SUBAPPLICATION mapping_AuxFunction2_IE (* Mapping for all AuxFunction2 *)
  (* Standard: 61499-2 *)
  (* Version 1.0, 2023-01-29, Franz *)
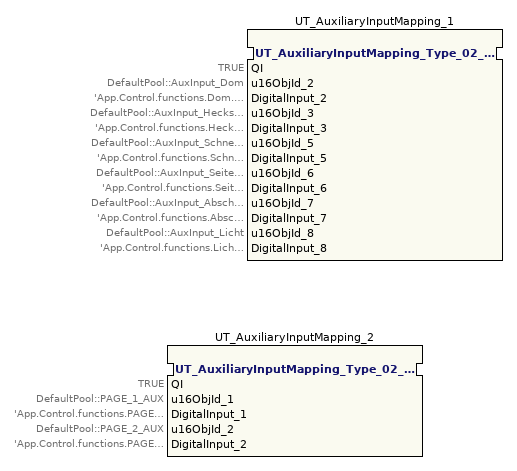
  FBS
    UT_AuxiliaryInputMapping_1 : UT_AuxiliaryInputMapping_Type_02_Bool_NonLatched_UP(QI := TRUE, u16ObjId_2 := DefaultPool::AuxInput_Dom, DigitalInput_2 := 'App.Control.functions.Dom.AuxInput', u16ObjId_3 := DefaultPool::AuxInput_Heckschieber, DigitalInput_3 := 'App.Control.functions.Heckschieber.AuxInput', u16ObjId_5 := DefaultPool::AuxInput_Schneidwerk, DigitalInput_5 := 'App.Control.functions.Schneidwerk.AuxInput', u16ObjId_6 := DefaultPool::AuxInput_Seitenschieber, DigitalInput_6 := 'App.Control.functions.Seitenschieber.AuxInput', u16ObjId_7 := DefaultPool::AuxInput_Abscheider, DigitalInput_7 := 'App.Control.functions.Abscheider.AuxInput', u16ObjId_8 := DefaultPool::AuxInput_Licht, DigitalInput_8 := 'App.Control.functions.Licht.AuxInput');
    UT_AuxiliaryInputMapping_2 : UT_AuxiliaryInputMapping_Type_02_Bool_NonLatched_UP(QI := TRUE, u16ObjId_1 := DefaultPool::PAGE_1_AUX, DigitalInput_1 := 'App.Control.functions.PAGES.PAGE_1.AUX', u16ObjId_2 := DefaultPool::PAGE_2_AUX, DigitalInput_2 := 'App.Control.functions.PAGES.PAGE_2.AUX');
  END_FBS
END_SUBAPPLICATION
